FUNCTION_BLOCK PtPreciseDiff
VAR_INPUT
	years: DINT;
    months: DINT;
    days: DINT;
    hours: DINT;
    minutes: DINT;
    seconds: DINT;
    microseconds: DINT;
    total_days: DINT;
END_VAR
VAR_OUTPUT
END_VAR
VAR
END_VAR

METHOD Set : BOOL
VAR_INPUT
	years: DINT;
    months: DINT;
    days: DINT;
    hours: DINT;
    minutes: DINT;
    seconds: DINT;
    microseconds: DINT;
    total_days: DINT;
END_VAR
THIS^.years := years;
THIS^.months := months;
THIS^.days := days;
THIS^.hours := hours;
THIS^.minutes := minutes;
THIS^.seconds := seconds;
THIS^.microseconds := microseconds;
THIS^.total_days := total_days;
END_METHOD

END_FUNCTION_BLOCK

(* stored: Version 1.1.0.1, ProductVersion 3.1.4024.12
   POU PtPreciseDiff: Id {685ddab2-ae24-41b4-8490-3b0ed69fc74d}, SpecialFunc None
   Method Set: Id {a7b02f8b-074a-44fd-a0c8-b7aee3edf92e} *)
